KUKA KRL data list: Pdetection.dat

&ACCESS RV2
&REL 970
&PARAM DISKPATH = KRC:\R1\Program\KukaMiling\Subprogs
DEFDAT  PDETECTION PUBLIC

DECL GLOBAL BOOL Nor1=TRUE
DECL GLOBAL BOOL Nor2=FALSE
DECL GLOBAL BOOL Nor3=TRUE
DECL GLOBAL BOOL Nor4=FALSE


DECL GLOBAL BOOL Nor5=TRUE
DECL GLOBAL BOOL Nor6=FALSE

DECL GLOBAL BOOL gbClk=TRUE

DECL GLOBAL BOOL gbSet1=FALSE
DECL GLOBAL BOOL gbSet2=FALSE
DECL GLOBAL BOOL gbSet3=FALSE
DECL GLOBAL BOOL gbSet4=FALSE

GLOBAL STRUC gP_Button BOOL actState
DECL GLOBAL gP_Button P_Button[6]
P_Button[1]={actState FALSE}

DECL BOOL lbMem=TRUE
ENDDAT
